Yaskawa INFORM job: 1PKT.JBI

/JOB
//NAME 1PKT
//POS
///NPOS 3,3,0,0,0,0
///TOOL 0
///POSTYPE ROBOT
///RECTAN
///RCONF 1,0,0,0,0,0,0,0,0,0,0,0,0,0,0,0,0,0,0,0,0,0,0,0
C00000=1391.737,-1304.065,-915.041,-88.1817,-0.6489,-1.7223
C00001=1392.033,-1404.912,-915.016,-88.1832,-0.6472,-1.7209
C00002=1391.737,-1304.065,-915.041,-88.1817,-0.6489,-1.7223
///RCONF 0,0,0,0,0,0,0,0,0,0,0,0,0,0,0,0,0,0,0,0,0,0,0,0
BC00000=592.196,3512.476,85.329
BC00001=592.196,3512.476,85.329
BC00002=592.196,3512.476,85.329
//INST
///DATE 2024/08/13 11:29
///ATTR SC,RW,RJ
////FRAME ROBOT
///GROUP1 RB1,BS1
NOP
MOVJ C00000 BC00000 VJ=5.00
MOVL C00001 BC00001 V=25.0  //1
MOVJ C00002 BC00002 VJ=5.00
END
